(* IEC 61131-3 sources: Elmo_Master/Lasal_PRG/MotionTCPDemo/Class/TCPCommunicationLogFilter, 1 file *)

(* ---- TCPCommunicationLogFilter.st ---- *)
(*!
<Class
	Name               = "TCPCommunicationLogFilter"
	Revision           = "1.0"
	RealtimeTask       = "false"
	CyclicTask         = "false"
	BackgroundTask     = "false"
	Sigmatek           = "true"
	OSInterface        = "false"
	HighPriority       = "false"
	Automatic          = "false"
	UpdateMode         = "Prescan"
	SharedCommandTable = "true"
	Objectsize         = "(530,120)"
	Comment            = "Derive class and overwrite Method CheckFilter() in order to filter logentries.">
	<Channels>
		<Server Name="ClassSvr" Visualized="false" Initialize="false" WriteProtected="true" Retentive="false" Comment="Derive Class and Connect Server to cLogFilter if logging entries shall be filtered."/>
	</Channels>
	<RevDoku>
		<Owner Company="Sigmatek" Author="HötAnt"/>
		<Dokumentation Revision="1.0" Date="2015-02-16" Author="ObeChr" Company="Sigmatek" Description="Prepared class for library."/>
		<Dokumentation Revision="1.0" Date="2014-04-17" Author="HötAnt" Company="Sigmatek" Description="Created class"/>
	</RevDoku>
</Class>
*)
TCPCommunicationLogFilter : CLASS
  //Servers:
	ClassSvr 	: SvrChCmd_DINT;
  //Clients:
  //Variables:
  //Functions:
				//! <Function Comment="Derive class and overwrite this method if you want the log entries to be filtered. Return FALSE if entry should be dropped, otherwise return TRUE." Name="CheckFilter"/>
	FUNCTION VIRTUAL GLOBAL CheckFilter
		VAR_INPUT
			pMNG_LogEntrie 	: ^TCPCommunication::t_s_LogEntry;
		END_VAR
		VAR_OUTPUT
			bAddToLog 	: BOOL;
		END_VAR;
  //Tables:
	FUNCTION @STD
		VAR_OUTPUT
			ret_code	: CONFSTATES;
		END_VAR;
	FUNCTION GLOBAL TAB @CT_;
END_CLASS;

#pragma using TCPCommunication

#pragma warning(disable:73);

FUNCTION VIRTUAL GLOBAL TCPCommunicationLogFilter::CheckFilter
	VAR_INPUT
		pMNG_LogEntrie 	: ^TCPCommunication::t_s_LogEntry;
	END_VAR
	VAR_OUTPUT
		bAddToLog 	: BOOL;
	END_VAR

  bAddToLog := TRUE;

END_FUNCTION
#pragma warning(default:73);
